{attribute 'GeneratedUsingTerminal: EJ2914-0000-0017'}
{attribute addProperty BoxType "EJ2914-0000-0017"}
{attribute addProperty Id "FSOEAT %I*FSOE_D94E700C6"}
{attribute addProperty CRC "365094833"}
{attribute addProperty Size "6"}
TYPE FSoE_Inputs_15C2E7B1 EXTENDS InputBase_8311D824 :
STRUCT
	{attribute addProperty Name "FSOE"}
	FSOE AT %I* : FSOE_D94E700C;
END_STRUCT
END_TYPE
